Universal Robots URScript: test2.script

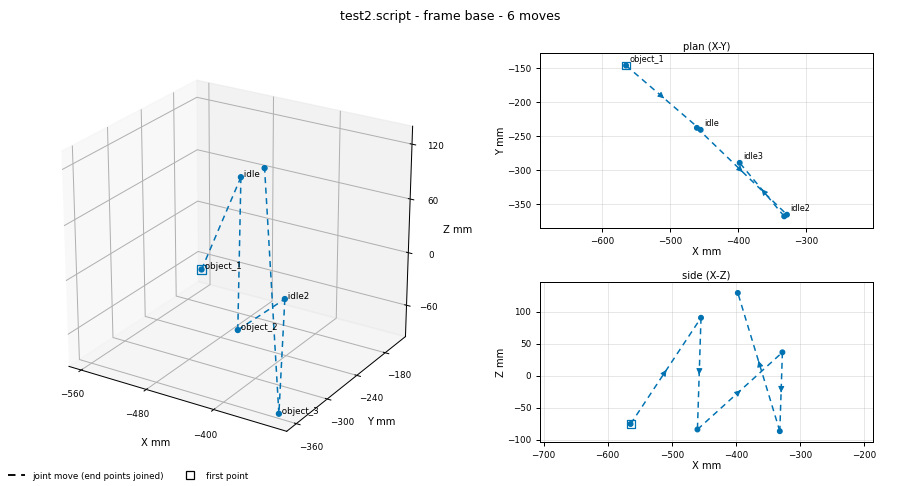
[picture p0: tool path of test2.script in frame base, 6 of 7 moves have a stored position in this frame; points joined in program order, loops and branches not executed]
def unnamed():
  set_safety_mode_transition_hardness(1)
  set_target_payload(1.500000, [0.000000, -0.002000, 0.046000], [0.003026, 0.003026, 0.003026, 0.000000, 0.000000, 0.000000])
  set_gravity([0.0, 0.0, 9.82])
  set_tcp(p[0.0,0.0,0.184,0.0,0.0,0.0])
  set_standard_analog_input_domain(0, 1)
  set_standard_analog_input_domain(1, 1)
  set_tool_analog_input_domain(0, 1)
  set_tool_analog_input_domain(1, 1)
  set_analog_outputdomain(0, 0)
  set_analog_outputdomain(1, 0)
  set_input_actions_to_default()
  set_tool_communication(False, 115200, 0, 1, 1.5, 3.5)
  set_tool_output_mode(0)
  set_tool_digital_output_mode(0, 1)
  set_tool_digital_output_mode(1, 1)
  set_tool_voltage(0)
  step_count_f83bf9cc_2243_44f5_a465_e855ca0bcf7d = 0.0
  thread Step_Counter_Thread_94936083_7f15_4ce7_8c00_c5da077e68f3():
    while (True):
      step_count_f83bf9cc_2243_44f5_a465_e855ca0bcf7d = step_count_f83bf9cc_2243_44f5_a465_e855ca0bcf7d + 1.0
      sync()
    end
  end
  run Step_Counter_Thread_94936083_7f15_4ce7_8c00_c5da077e68f3()
  global Line_1=p[0.0,0.0,0.0,0.0,0.0,0.0]
  global Line_2=p[0.0,0.0,0.0,0.0,0.0,0.0]
  global Plane_1=p[-0.361487432735338,-0.016717979378191757,0.10394933298158474,0.8032803749589464,-1.48273794275507,-1.3712545351254601]
  global Plane_2=p[-0.4390181010417212,-0.5025363244384129,0.07754186088006663,0.0242452931196319,-0.008431548293163078,-0.5708956925038724]
  global Plane_3=p[-0.25480483753173705,-0.5081372437231373,0.07201538765959875,-9.039930063647936E-5,-1.434349324572951E-4,-0.3090720642039013]
  global Point_3=p[0.0,0.0,0.0,0.0,0.0,0.0]
  global floorgripper=p[-0.2464960731348849,-0.4897452928079739,0.0709944577944641,1.7320762453741406E-4,5.47703051263464E-6,-0.32694642097279897]
  global front_collision=p[-0.4941642762715196,-0.6127463334128198,0.7662532960153384,1.5,4.484756383203096E-16,2.3363997805214006E-16]
  global table=p[-0.8492357722348507,-0.0703668253590126,-0.04045,-2.900828785048298,-1.2031999063950631,-7.106365334326772E-4]
  # begin: URCap Installation Node
  #   Source: External Control, 1.0.5, FZI Research Center for Information Technology
  #   Type: External Control
  # end: URCap Installation Node
  global object_1_p=p[-.564243275223, -.145996988541, -.075050811661, 1.235769180818, 2.851309869901, -.020353683024]
  global object_1_q=[0.008059142157435417, -0.9971593779376526, 1.9021952787982386, -2.4488874874510707, -1.5439637343036097, -0.7457745710956019]
  global idle_p=p[-.454486621211, -.240538631491, .090530219108, -1.199706015407, -2.864351512455, .017036689035]
  global idle_q=[0.23056091368198395, -1.4333766561797638, 2.0075834433185022, -2.179491182366842, -1.5816033522235315, -0.5485928694354456]
  global object_2_p=p[-.460057510970, -.237656426558, -.083616600867, -1.200206705239, -2.869460532865, -.018746999897]
  global object_2_q=[0.23110152781009674, -1.0798893135837098, 2.1245697180377405, -2.6324688396849574, -1.5972779432879847, -0.5480869452105921]
  global idle2_p=p[-.327612513548, -.365336542712, .036682236756, -1.159750334070, -2.868952863758, .074729301342]
  global idle2_q=[0.5696951150894165, -1.4080671978047867, 2.162783924733297, -2.390435834924215, -1.5787137190448206, -0.2343199888812464]
  global object_3_p=p[-.331659758824, -.367783220054, -.086289276566, 1.175406119521, 2.907611741346, .035654001680]
  global object_3_q=[0.5686042904853821, -1.1019612711719056, 2.161781136189596, -2.6078878841795863, -1.5780423323260706, -0.2343080679522913]
  global idle3_p=p[-.397101045856, -.289093386097, .129218364448, 1.150366212970, 2.822106084839, .015705950974]
  global idle3_q=[0.3212403357028961, -1.487023004596569, 1.9256628195392054, -1.9299866161742152, -1.5162485281573694, -0.4793055693255823]
  $ 1 "BeforeStart"
  $ 2 "Home"
  movej([-0.2136619726764124, -1.4704142820886155, 1.4500101248370567, -1.5527248562178393, -1.6063321272479456, -1.7763568394002505E-15], a=1.3962634015954636, v=1.0471975511965976)
  while (True):
    $ 3 "Robot Program"
    $ 4 "MoveJ"
    $ 5 "Wait DI[0]=HI"
    while (get_standard_digital_in(0) == False):
      sync()
    end
    $ 6 "object_1" "breakAfter"
    movej(get_inverse_kin(object_1_p, qnear=object_1_q), a=1.3962634015954636, v=1.0471975511965976)
    $ 7 "idle" "breakAfter"
    movej(get_inverse_kin(idle_p, qnear=idle_q), a=1.3962634015954636, v=1.0471975511965976)
    $ 8 "object_2" "breakAfter"
    movej(get_inverse_kin(object_2_p, qnear=object_2_q), a=1.3962634015954636, v=1.0471975511965976)
    $ 9 "idle2" "breakAfter"
    movej(get_inverse_kin(idle2_p, qnear=idle2_q), a=1.3962634015954636, v=1.0471975511965976)
    $ 10 "object_3" "breakAfter"
    movej(get_inverse_kin(object_3_p, qnear=object_3_q), a=1.3962634015954636, v=1.0471975511965976)
    $ 11 "idle3" "breakAfter"
    movej(get_inverse_kin(idle3_p, qnear=idle3_q), a=1.3962634015954636, v=1.0471975511965976)
    $ 12 "Set DO[0]=On"
    set_standard_digital_out(0, True)
  end
end
